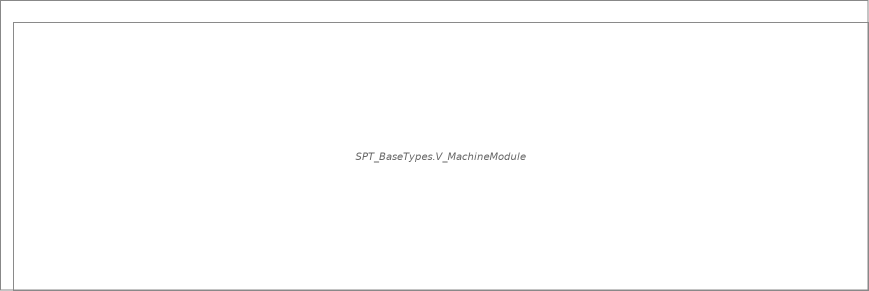
VISUALIZATION Visualization  // 869x291
    Frame (13,22 856x269)
        shows SPT_BaseTypes.V_MachineModule(HMI := MAIN.Machine.PackMLBaseModule_HMI)
END_VISUALIZATION

(* stored: Version 1.1.0.1, ProductVersion 3.1.4024.12
   Visu Visualization: Id {5be74494-91dd-4b66-826f-b48c7fe0c03b} *)
